PROGRAM P_ADSCommManager
VAR // comm values
	bValueToWrite		:	BOOL;
	bAutoWriteNewVal	:	BOOL;
	bWriteNewValOnce	:	BOOL;
	bCurrentValue		:	BOOL;
	sVarName			:	STRING(255) := 'P_Kuchnia._fbHeater_0.bManualValveOpen';
END_VAR
VAR
	fbWrite				:	FB_WriteAdsSymByName;
	fbRead				:	FB_ReadAdsSymByName;
	fbRTrigWriteOnce	:	R_TRIG;
	fbTonAutoWrite		:	TON := (pt := T#1S);
	iSwitch				:	INT := 1;
	bWriteInProgress	:	BOOL;
END_VAR

fbRTrigWriteOnce(clk := bWriteNewValOnce);
fbTonAutoWrite(IN := NOT fbTonAutoWrite.Q);
IF bAutoWriteNewVal OR fbread.bBusy THEN
	CASE iSwitch OF 
		1:
			IF fbTonAutoWrite.Q THEN
				fbRead(bRead := TRUE,
					sVarName := sVarName,
					nDestAddr := ADR(bCurrentValue),
					nLen := SIZEOF(bcurrentValue));
			END_IF
			fbRead();
			IF NOT fbRead.bBusy	AND NOT fbRead.bError THEN
				fbRead(bRead := FALSE);
				iSwitch := 2;
			END_IF
		2:
			IF bCurrentValue <> bValueToWrite THEN
				fbWrite(bWrite := TRUE,
					sVarName := sVarName,
					nSrcAddr := ADR(bValueToWrite),
					nlen := SIZEOF(bValueToWrite));
				IF NOT fbWrite.bBusy AND  NOT fbWrite.bError THEN
					fbWrite(bWrite := FALSE);
					iSwitch := 1;
				END_IF
			END_IF
	END_CASE
END_IF
IF fbRTrigWriteOnce.Q OR bWriteInProgress THEN
	fbWrite(bWrite := TRUE,
					sVarName := sVarName,
					nSrcAddr := ADR(bValueToWrite),
					nlen := SIZEOF(bValueToWrite));
	bWriteInProgress := TRUE;
	IF NOT fbWrite.bBusy AND  NOT fbWrite.bError THEN
		fbRead(bRead := TRUE,
			sVarName := sVarName,
			nDestAddr := ADR(bCurrentValue),
			nLen := SIZEOF(bcurrentValue));
		IF NOT fbRead.bBusy	AND NOT fbRead.bError THEN
			fbRead(bRead := FALSE);
			fbWrite(bWrite := FALSE);
			bWriteInProgress := FALSE;
		END_IF
	END_IF
END_IF

METHOD FB_init : BOOL
VAR_INPUT
	bInitRetains : BOOL := FALSE; // if TRUE, the retain variables are initialized (warm start / cold start)
	bInCopyCode : BOOL := FALSE;  // if TRUE, the instance afterwards gets moved into the copy code (online change)
END_VAR
fbRead.eComMode := E_AdsComMode.eAdsComModeFastCom;
fbRead.sNetId := '5.21.22.214.1.1';
fbRead.nPort := 851;
fbWrite.eComMode := E_AdsComMode.eAdsComModeFastCom;
fbWrite.sNetId := '5.21.22.214.1.1';
fbWrite.nPort := 851;
END_METHOD

END_PROGRAM

(* stored: Version 1.1.0.1, ProductVersion 3.1.4024.9
   POU P_ADSCommManager: Id {01ba0257-6e6b-4545-ad25-02ccef70045c}, SpecialFunc None
   Method FB_init: Id {c17cece7-f1a0-46bb-bec9-71ca8f046656} *)
